FUNCTION_BLOCK FB_CheckMessageBounds
VAR_IN_OUT
	
	iqArrayToCheck:typeMessage; //type of message bounds
	iqPassThruMessageStart:INT; //pass to /from alarm to warning start, warnings listed after all alarms
	
	//
	//new message rows using table
	qSpecialMsgRows:ARRAY[1..gHMIDataConst.gNumberOfMessagesScreen] OF typeNewMsg;
	qSpecialMsgRowsStyle:ARRAY[1..gHMIDataConst.gNumberOfMessagesScreen] OF typeNewMsgStyle;
	
	//messages were changed, update list
	iqMsgChangeUpdateList:BOOL;
	
	
END_VAR
VAR_OUTPUT
	qAnyMsgActive: BOOL;
	qMsgNumberActive: UINT;
	
	qSingleMessage: STRING(255);
	
	qAllMessages: STRING;
	
	//declare, follows typeMessageRowsArry
	qMsgRows:ARRAY[1..gHMIDataConst.gNumberOfMessagesScreen] OF typeMessageRow;
	
	
	
	
	

END_VAR
VAR
	i: INT;//for the loop
	lowestValue: UDINT :=4294967295; //set as init for highest possible value and work down from there
	lowestMessage: INT;
	allstrings: STRING;
	rollinglowestValue: UDINT :=0; //set as init for lowest possible value and work up
	newlineInsert: string;

	messageHeader: STRING(255);
	memcomparecheck: DINT;
	memchanged: BOOL;
	messagenum: UINT;
	strheader:STRING(255);
	
	n: UINT;
	returnclearing: UDINT;
	msgIndex: INT;
	timWaitDelay: TON;
	
	rollingOffset:INT; //offset for injecting further messages
	k: UINT;
	strlengtest: INT;
	tWarnOffset:INT; //starting location for warning
	timPulseChange: TP;
	timPulseChangedMessage: TP;
	j: INT;
	a: UINT;
END_VAR

VAR_INPUT
	iMessageGroup: UINT;
	isAlarm: BOOL; //for colour assigment
	isWarning: BOOL; //for colour assigment




END_VAR
VAR // added by the converter: edge detectors and wires of the graphical bodies
    _rt1 : R_TRIG;
END_VAR

// Reset before scan
actArraysMatch();
actPassMessageChange();

IF memchanged OR iqMsgChangeUpdateList THEN 
    // Reset status variables
    qAnyMsgActive := FALSE;
    qMsgNumberActive := 0;  
    actCleanDownMsg();
    
    lowestValue := 4294967295;
    lowestMessage := 0;
    rollinglowestValue := 0;
    allstrings := '';

    // FIRST PASS: Determine active status and find the oldest (lowest timestamp) message
    FOR i := 0 TO GlobalMessages.gNumMessagesPerType - 1 DO
        IF iqArrayToCheck.message[i] THEN
            qAnyMsgActive := TRUE;
            qMsgNumberActive := INT_TO_UINT(i);
            
            // Assign CycleCount timestamp if it's a brand new activation
            IF NOT iqArrayToCheck.messageActive[i] AND iqArrayToCheck.messageTimeActive[i] = 0 THEN
                iqArrayToCheck.messageTimeActive[i] := System.myPlcInfoTask1.CycleCount;
            END_IF
            
            // Check chronological order (looking for oldest timestamp > 1)
            IF iqArrayToCheck.messageTimeActive[i] > 1 AND iqArrayToCheck.messageTimeActive[i] < lowestValue THEN
                lowestValue := iqArrayToCheck.messageTimeActive[i];
                lowestMessage := i;                                 
                qSingleMessage := iqArrayToCheck.text[i];           
            END_IF
        ELSE
            // Reset message tracking states cleanly if cleared
            IF iqArrayToCheck.messageActive[i] THEN
                iqArrayToCheck.messageActive[i] := FALSE;
                iqArrayToCheck.messageTimeActive[i] := 0;
            END_IF
        END_IF
    END_FOR;

    // Handle global state if no messages are found
    IF NOT qAnyMsgActive THEN
        qSingleMessage := 'no message';
        lowestMessage := 0;
        lowestValue := 4294967295;
        rollinglowestValue := 0;
        qAllMessages := '';
    ELSE
        rollinglowestValue := lowestValue;
    END_IF

    // SECOND PASS: Only construct strings and handle active logic shifts if warnings/alarms exist
    IF qAnyMsgActive AND rollinglowestValue >= 0 THEN
        FOR i := 0 TO GlobalMessages.gNumMessagesPerType - 1 DO
            IF iqArrayToCheck.message[i] THEN
                // Combine strings efficiently inside the conditional change event
                newlineInsert := concat(iqArrayToCheck.text[i], '$0D'); 
                messagenum := iMessageGroup + INT_TO_UINT(i); 
                strheader := concat(DINT_TO_STRING(messagenum), ' '); 
                newlineInsert := concat(strheader, newlineInsert);
                allstrings := concat(newlineInsert, allstrings); 
                
                iqArrayToCheck.messageActive[i] := TRUE;
            END_IF
        END_FOR;
        qAllMessages := allstrings;
    END_IF

    // THIRD PASS: Populate HMI Row Data arrays safely (Fixing out-of-bounds boundary)
    msgindex := 1;
    IF isWarning THEN
        tWarnOffset := iqPassThruMessageStart;
        actClearDownExcessWarn(); 
    ELSE
        tWarnOffset := 0;
    END_IF

    IF isAlarm AND NOT qAnyMsgActive THEN
        iqPassThruMessageStart := 0;
    END_IF

    FOR i := 0 TO GlobalMessages.gNumMessagesPerType - 1 DO // FIXED: Added "- 1" to prevent CPU crash
        IF iqArrayToCheck.messageActive[i] THEN
            qMsgRows[msgindex].msgText := iqArrayToCheck.text[i];
            qSpecialMsgRows[msgindex + tWarnOffset].text := iqArrayToCheck.text[i];
            qSpecialMsgRows[msgindex + tWarnOffset].timeRaised := UDINT_TO_STRING(iqArrayToCheck.messageTimeActive[i]);
            
            // Styling logic definitions
            IF isAlarm THEN
                qMsgRows[msgindex].isAlarm := TRUE;
                qMsgRows[msgindex].isWarning := FALSE;
                qSpecialMsgRowsStyle[msgindex + tWarnOffset].colourToApply := HMIColour.colourRed;
                qSpecialMsgRowsStyle[msgindex + tWarnOffset].isColoured := TRUE;
            ELSIF isWarning THEN
                qMsgRows[msgindex].isAlarm := FALSE;
                qMsgRows[msgindex].isWarning := TRUE;
                qSpecialMsgRowsStyle[msgindex + tWarnOffset].colourToApply := HMIColour.colourYellow;
                qSpecialMsgRowsStyle[msgindex + tWarnOffset].isColoured := TRUE;
            ELSE
                qMsgRows[msgindex].isAlarm := FALSE;
                qMsgRows[msgindex].isWarning := FALSE;
                qSpecialMsgRowsStyle[msgindex + tWarnOffset].colourToApply := HMIColour.colourGreyBackground;
                qSpecialMsgRowsStyle[msgindex + tWarnOffset].isColoured := FALSE;
            END_IF
            
            IF qSpecialMsgRows[msgindex].text = '' THEN
                qSpecialMsgRows[msgindex].timeRaised := '';
            END_IF
            
            msgindex := msgindex + 1;
            IF msgindex > GlobalMessages.gNumMessagesPerType - 1 THEN
                EXIT;
            END_IF
        END_IF
    END_FOR;
    
    // Calculate display offsets only on mutation, removing the continuous "OR TRUE" scan loop
    rollingOffset := 0;
    IF isAlarm THEN
        FOR k := 1 TO gHMIDataConst.gNumberOfMessagesScreen DO
            // Efficient replacement for expensive LEN() functions
            IF qSpecialMsgRows[k].text <> '' AND qSpecialMsgRowsStyle[k].colourToApply = HMIColour.colourRed THEN
                rollingOffset := UINT_TO_INT(k);
                iqPassThruMessageStart := rollingOffset;        
            END_IF
        END_FOR;
    END_IF

END_IF; // End of Event Execution Block

// Warning tracking state check remains live to handle background UI logic triggers
IF qAnyMsgActive AND isWarning AND qSpecialMsgRowsStyle[tWarnOffset + 1].colourToApply <> HMIColour.colourYellow THEN
    iqMsgChangeUpdateList := TRUE;
ELSE
    IF isWarning THEN iqMsgChangeUpdateList := FALSE; END_IF
END_IF;

ACTION actArraysMatch:
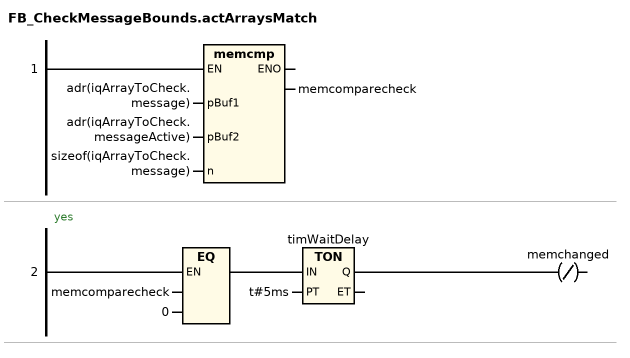
// NETWORK 1
memcomparecheck := memcmp(pBuf1 := adr(iqArrayToCheck.message), pBuf2 := adr(iqArrayToCheck.messageActive), n := sizeof(iqArrayToCheck.message));

// NETWORK 2
// yes
timWaitDelay(IN := memcomparecheck = 0, PT := t#5ms); // TON
memchanged := NOT timWaitDelay.Q;
END_ACTION

ACTION actCleanDownMsg:
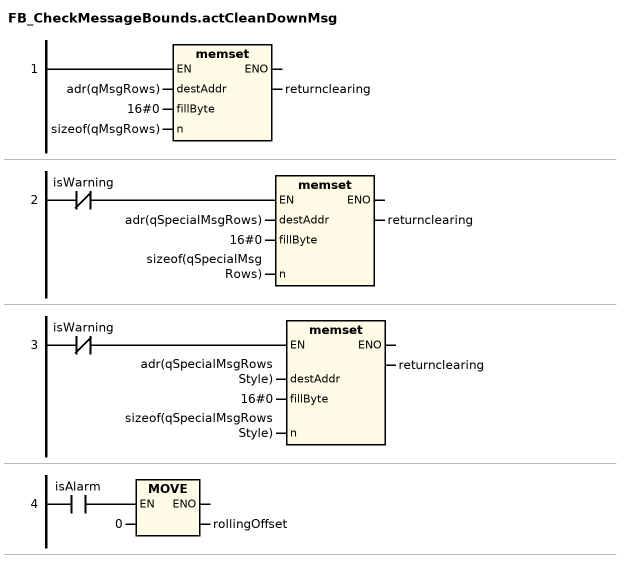
// NETWORK 1
returnclearing := memset(destAddr := adr(qMsgRows), fillByte := 16#0, n := sizeof(qMsgRows));

// NETWORK 2
IF NOT isWarning THEN
    returnclearing := memset(destAddr := adr(qSpecialMsgRows), fillByte := 16#0, n := sizeof(qSpecialMsgRows));
END_IF

// NETWORK 3
IF NOT isWarning THEN
    returnclearing := memset(destAddr := adr(qSpecialMsgRowsStyle), fillByte := 16#0, n := sizeof(qSpecialMsgRowsStyle));
END_IF

// NETWORK 4
IF isAlarm THEN rollingOffset := 0; END_IF
END_ACTION

ACTION actClearDownExcessWarn:

//clear down warning messages after last alarm message
//FOR j:= tWarnOffset + 1 TO GlobalMessages.gNumMessagesPerType DO
FOR j:= tWarnOffset + 1 TO UINT_TO_INT(gHMIDataConst.gNumberOfMessagesScreen) DO
 qSpecialMsgRowsStyle[j].colourToApply := HMIColour.colourGreyBackground;
 qSpecialMsgRowsStyle[j].isColoured := FALSE;
 qSpecialMsgRows[j].text := '';
END_FOR
END_ACTION

ACTION actPassMessageChange:
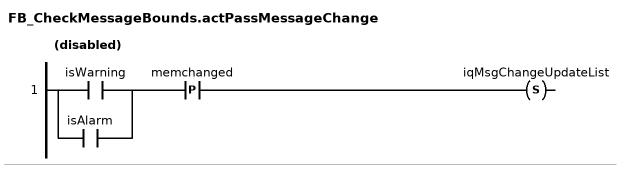
// NETWORK 1 (disabled)
// _rt1(CLK := memchanged);
// iqMsgChangeUpdateList S= (isWarning OR isAlarm) AND _rt1.Q;
END_ACTION

END_FUNCTION_BLOCK

(* stored: Version 1.1.0.1, ProductVersion 3.1.4024.11
   POU FB_CheckMessageBounds: Id {cfd3e64b-34a3-43a4-b491-e0f565bbe474}, SpecialFunc None
   Action actArraysMatch: Id {deaf4cea-369a-4b23-adf0-691b3612839c}
   Action actCleanDownMsg: Id {c459896b-96a2-4e11-8e93-84fa94812ca5}
   Action actClearDownExcessWarn: Id {101dc8f4-d8c6-4be9-bb79-5924a7d90678}
   Action actPassMessageChange: Id {d6737f3f-2922-49a8-82a5-cbae2265c9fc} *)
